(* Logix 5000 project; controller WWTP_SEC_CLX vendor 1 type 14 code 54 rev 17.2; software revision 17.00; part 10 of 13 *)
(* tags used below, declared in another part *)
   Inp_SpeedFdbk : INT;   // Speed Feedbak in Drive Units (typ. 0-32767 = 0 to max freq.)
   Inp_Datalink : INT;   // Auxiliary Signal (datalink) Input in Drive (raw) Units
   Inp_Ready : BOOL;   // 1=Drive is ready to run
   Inp_CommandDir : BOOL;   // 1=Drive is commanded Forward, 0=Drive is commanded Reverse
   Inp_ActualDir : BOOL;   // 1=Drive is running Forward, 0=Drive is running Reverse
   Inp_Accelerating : BOOL;   // 1=Drive is accelerating
   Inp_Decelerating : BOOL;   // 1=Drive is decelerating
   Inp_Alarm : BOOL;   // 1=Drive has an Alarm Condition (see drive display or manual)
   Inp_Faulted : BOOL;   // 1=Drive has Faulted (see drive display or manual)
   Inp_AtSpeed : BOOL;   // 1=Drive is at commanded speed
   Inp_FwdPermOK : BOOL;   // 1=Permissives OK, drive can start Forward
   Inp_FwdNBPermOK : BOOL;   // 1=Non-Bypassable Permissives OK, drive can start Forward
   Inp_RevPermOK : BOOL;   // 1=Permissives OK, drive can start Reverse
   Inp_RevNBPermOK : BOOL;   // 1=Non-Bypassable Permissives OK, motor can start Reverse
   Inp_IntlkOK : BOOL;   // 1=Interlocks OK, drive can start/run
   Inp_NBIntlkOK : BOOL;   // 1=Non-Bypassable Interlocks OK, drive can start/run
   Inp_IOFault : BOOL;   // Input Communication Status 0=OK, 1=fail
   Inp_Sim : BOOL;   // 1=Simulate working drive; 0=Start/Stop/ Monitor actual drive
   Cfg_HasReverse : BOOL;   // 1=Drive can be run reverse, 0=Forward only
   Cfg_HasJog : BOOL;   // 1=Drive Jog Command enabled/visible, 0=Drive Jog Command not allowed
   Cfg_UseRunFdbk : BOOL;   // 1=Drive run feedback should be used for failure checking
   Cfg_HasInpDatalink : BOOL;   // 1=A signal is connected to Inp_Datalink1
   Cfg_HasOutDatalink : BOOL;   // 1=A signal is connected to Out_Datalink1
   Cfg_SetTrack : BOOL;   // 1=PSets track OSets in Oper, OSets track PSets in Prog, 0=no tracking
   Cfg_SetTrackOvrdHand : BOOL;   // 1=Prog/Oper Settings track Override/Hand speed reference
   Cfg_PCmdClear : BOOL;   // 1=Clear Program Commands on receipt 0=Leave Set
   Cfg_SpeedFdbkRawMin : INT;   // Speed Feedback Minimum in Drive (raw) Units (for scaling)
   Cfg_SpeedFdbkRawMax : INT;   // Speed Feedback Maximum in Drive (raw) Units (for scaling)
   Cfg_SpeedFdbkEUMin : REAL;   // Speed Feedback Minimum in Engineering Units (for scaling)
   Cfg_SpeedFdbkEUMax : REAL;   // Speed Feedback Maximum in Engineering Units (for scaling)
   Cfg_InpDatalinkRawMin : INT;   // Input Datalink Minimum in Drive (raw) Units (for scaling)
   Cfg_InpDatalinkRawMax : INT;   // Input Datalink Maximum in Drive (raw) Units (for scaling)
   Cfg_InpDatalinkEUMin : REAL;   // Input Datalink Minimum in Engineering Units (for scaling)
   Cfg_InpDatalinkEUMax : REAL;   // Input Datalink Maximum in Engineering Units (for scaling)
   PSet_SpeedRef : REAL;   // Program Setting of Speed Reference (EU)
   PSet_Owner : DINT;   // Program Owner Request ID (non-zero) or Release (zero)
   OSet_SpeedRef : REAL;   // Operator Setting of Speed Reference (EU)
   PCmd_Start : BOOL;   // Program Command to Start Drive
   PCmd_Stop : BOOL;   // Program Command to Stop Drive
   PCmd_Fwd : BOOL;   // Program Command to set direction to Fowrard
   PCmd_Rev : BOOL;   // Program Command to set direction to Reverse
   PCmd_Acq : BOOL;   // Program Command to Acquire ownership (Oper/OOS to Prog)
   PCmd_Rel : BOOL;   // Program Command to Release ownership (Prog to OOS)
   PCmd_Lock : BOOL;   // Program Command to Lock Mode in Prog
   PCmd_Unlock : BOOL;   // Program Command to Unlock Mode
   PCmd_Reset : BOOL;   // Program Command to Reset drive fault and all Alarms requiring Reset
   PCmd_FailToStartInhibit : BOOL;   // Program Command to Inhibit Fail to Start Alarm
   PCmd_FailToStartUninhibit : BOOL;   // Program Command to Uninhibit Fail to Start Alarm
   PCmd_FailToStopInhibit : BOOL;   // Program Command to Inhibit Fail to Stop Alarm
   PCmd_FailToStopUninhibit : BOOL;   // Program Command to Uninhibit Fail to Stop Alarm
   PCmd_IntlkTripInhibit : BOOL;   // Program Command to Inhibit Interlock Trip Alarm
   PCmd_IntlkTripUninhibit : BOOL;   // Program Command to Uninhibit Interlock Trip Alarm
   PCmd_DriveFaultInhibit : BOOL;   // Program Command to Inhibit Drive Fault Alarm
   PCmd_DriveFaultUninhibit : BOOL;   // Program Command to Uninhibit Drive Fault Alarm
   PCmd_IOFaultInhibit : BOOL;   // Program Command to Inhibit I/O Fault Alarm
   PCmd_IOFaultUninhibit : BOOL;   // Program Command to Uninhibit I/O Fault Alarm
   OCmd_Start : BOOL;   // Operator Command to Start Drive
   OCmd_Stop : BOOL;   // Operator Command to Stop Drive
   OCmd_Jog : BOOL;   // Operator Command to Jog Drive (not cleared by P_VSD!)
   OCmd_Fwd : BOOL;   // Operator Command to set direction to Forward
   OCmd_Rev : BOOL;   // Operator Command to set direction to Reverse
   OCmd_Bypass : BOOL;   // Operator Command to Bypass all Bypassable Interlocks and Permissives
   OCmd_Check : BOOL;   // Operator Command to Check (not bypass) all Interlocks and Permissives
   MCmd_Disable : BOOL;   // Maintenance Command to Disable Drive
   MCmd_Enable : BOOL;   // Maintenance Command to Enable (allow to run) Drive
   OCmd_Reset : BOOL;   // Operator Command to Reset all Alarms requiring Reset
   Val_SpeedRef : REAL;   // Speed Reference (target) to drive
   Val_SpeedFdbk : REAL;   // Speed Feedback (actual) from drive
   Val_InpDatalink : REAL;   // Input Datalink value from drive
   Val_OutDatalink : REAL;   // Output Datalink value to drive
   Val_SpeedFdbkEUMin : REAL;   // Minimum of Speed Feedback = MIN (Cfg_SpeedFdbkEUMin, Cfg_SpeedFdbkEUMax)
   Val_SpeedFdbkEUMax : REAL;   // Maximum of Speed Feedback = MAX (Cfg_SpeedFdbkEUMin, Cfg_SpeedFdbkEUMax)
   Val_Owner : DINT;   // Current Object Owner ID (0=not owned)
   Val_Notify : SINT;   // Current Alarm Level and Acknowledgement (enumeration)
   Sts_Stopped : BOOL;   // 1=Drive requested to stop and is confirmed stopped
   Sts_Starting : BOOL;   // 1=Drive requested to run and awaiting run feedback
   Sts_Running : BOOL;   // 1=Drive requested to run and is confirmed running
   Sts_Stopping : BOOL;   // 1=Drive requested to stop and awaiting stopped feedback
   Sts_Jogging : BOOL;   // 1=Drive requested to Jog
   Sts_CommandDir : BOOL;   // 1=Drive commanded to Forward, 0=Reverse
   Sts_ActualDir : BOOL;   // 1=Drive Actual direction is Forward, 0=Reverse
   Sts_Accel : BOOL;   // 1=Drive is Accelerating
   Sts_Decel : BOOL;   // 1=Drive is Decelerating
   Sts_NotReady : BOOL;   // 1=Drive is Not Ready (cannot be started) Check alarms, stops, faults
   Sts_Alarm : BOOL;   // 1=Drive has an Alarm (see drive display or manual)
   Sts_AtSpeed : BOOL;   // 1=Drive is running at reference speed
   Sts_Available : BOOL;   // 1=Drive available for control by automation (Prog)
   Sts_Bypass : BOOL;   // 1=Bypassable Interlocks and Permissives are Bypassed
   Sts_Disabled : BOOL;   // 1=Drive is Disabled
   Sts_Hand : BOOL;   // 1=Mode is Hand (supersedes Maint, Ovrd, Prog, Oper)
   Sts_Maint : BOOL;   // 1=Mode is Maintenance (supersedes Ovrd, Prog, Oper)
   Sts_Ovrd : BOOL;   // 1=Mode is Override (supersedes Prog, Oper)
   Sts_Prog : BOOL;   // 1=Mode is Program (auto)
   Sts_Oper : BOOL;   // 1=Mode is Operator (manual)
   Sts_FailToStop : BOOL;   // 1=Drive Failed to Stop
   Rdy_Start : BOOL;   // 1=Ready to receive OCmd_Start (enables HMI button)
   Rdy_Stop : BOOL;   // 1=Ready to receive OCmd_Stop (enables HMI button)
   Rdy_Jog : BOOL;   // 1=Ready to receive OCmd_Jog (enables HMI button)
   Rdy_Fwd : BOOL;   // 1=Ready to receive OCmd_Fwd (enabled HMI button)
   Rdy_Rev : BOOL;   // 1=Ready to receive OCmd_Rev (enables HMI button)
   Rdy_Bypass : BOOL;   // 1=Ready to receive OCmd_Bypass (enables HMI button)
   Rdy_Check : BOOL;   // 1=Ready to receive OCmd_Check (enables HMI button)
   Rdy_Disable : BOOL;   // 1=Ready to receive MCmd_Disable (enables HMI button)
   Rdy_Enable : BOOL;   // 1=Ready to receive MCmd_Enable (enables HMI button)
   Rdy_Reset : BOOL;   // 1=Ready to receive OCmd_Reset (enables HMI button)
   Mode : P_Mode;   // Drive Mode Selection
   IOFault : P_Alarm;   // I/O Fault Alarm
   IntlkTrip : P_Alarm;   // Interlock Trip Alarm
   FailToStop : P_Alarm;   // Drive Failed to Stop Alarm
   FailToStart : P_Alarm;   // Drive Failed to Start Alarm
   Wrk_Run : BOOL;   // 1=Drive should be "running", 0=should be "stopped"
   Wrk_AccelT : TIMER;   // Simulation Accel Ramp timer until Running at speed
   Wrk_Fault : BOOL;   // 1=any Fault has been detected
   Wrk_DecelT : TIMER;   // Simulation Decel Ramp time until fully stopped
   Wrk_RunFdbk : BOOL;   // Run Feedback based on mode, simulation, etc. 1=running
   Wrk_Notify : DINT;   // Buffer for building Val_Notify
   Wrk_Bypass : BOOL;   // Internal Bypassable Permissives and Interlocks are Bypassed flag
   Wrk_Disabled : BOOL;   // Internal Drive is Disabled
   DriveFault : P_Alarm;   // Drive Faulted Alarm
   Wrk_SpeedRef : REAL;   // Working copy of Speed Reference (for limiting)
   Wrk_Rev : BOOL;   // Working (internal) Direction 1=Reverse 0=Forward (default)
   Wrk_Jog : BOOL;   // 1=Jog Drive, 0=Drive not jogging
   Wrk_OutDatalink : REAL;   // Selected Output Datalink setting
(* P_VSD, continued *)

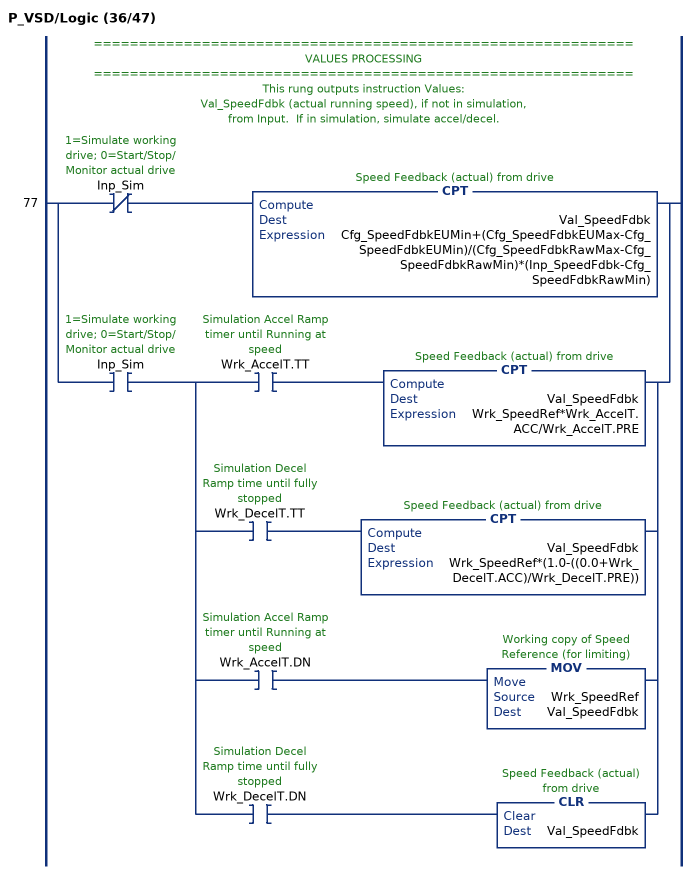
   // ============================================================
   // VALUES PROCESSING
   // ============================================================
   // This rung outputs instruction Values:
   // Val_SpeedFdbk (actual running speed), if not in simulation,
   // from Input.  If in simulation, simulate accel/decel.
   77: [XIO(Inp_Sim) CPT(Val_SpeedFdbk,Cfg_SpeedFdbkEUMin+(Cfg_SpeedFdbkEUMax-Cfg_SpeedFdbkEUMin)/(Cfg_SpeedFdbkRawMax-Cfg_SpeedFdbkRawMin)*(Inp_SpeedFdbk-Cfg_SpeedFdbkRawMin)) ,XIC(Inp_Sim) [XIC(Wrk_AccelT.TT) CPT(Val_SpeedFdbk,Wrk_SpeedRef*Wrk_AccelT.ACC/Wrk_AccelT.PRE) ,XIC(Wrk_DecelT.TT) CPT(Val_SpeedFdbk,Wrk_SpeedRef*(1.0-((0.0+Wrk_DecelT.ACC)/Wrk_DecelT.PRE))) ,XIC(Wrk_AccelT.DN) MOV(Wrk_SpeedRef,Val_SpeedFdbk) ,XIC(Wrk_DecelT.DN) CLR(Val_SpeedFdbk) ] ];
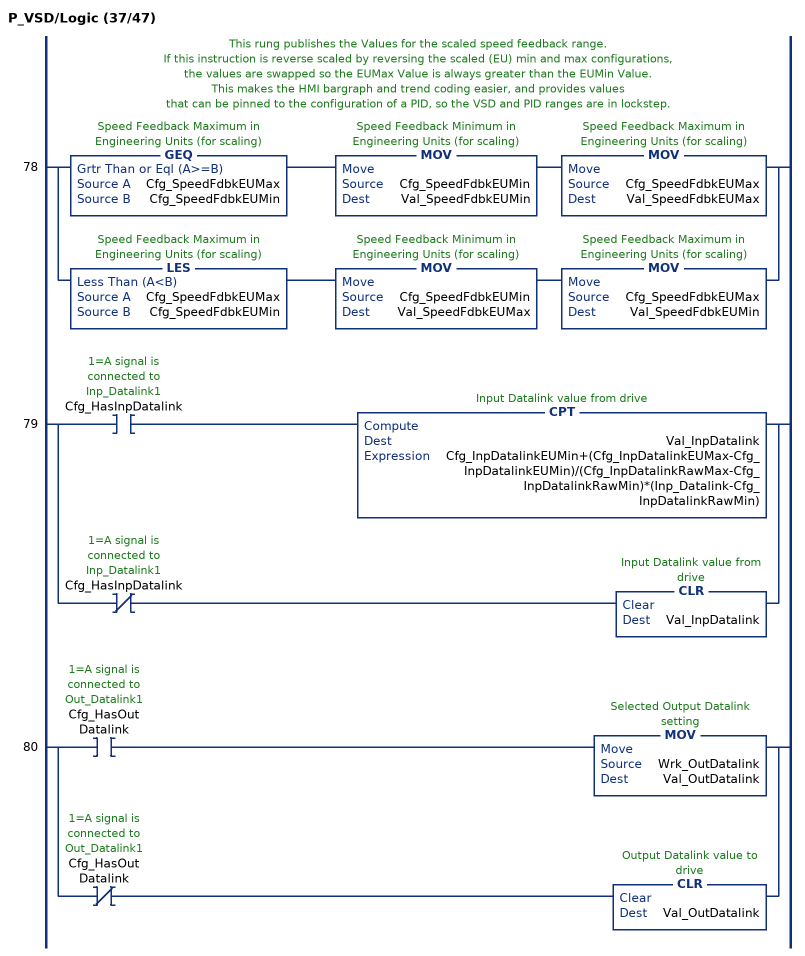
   // This rung publishes the Values for the scaled speed feedback range.
   // If this instruction is reverse scaled by reversing the scaled (EU) min and max configurations,
   // the values are swapped so the EUMax Value is always greater than the EUMin Value.
   // This makes the HMI bargraph and trend coding easier, and provides values
   // that can be pinned to the configuration of a PID, so the VSD and PID ranges are in lockstep.
   78: [GEQ(Cfg_SpeedFdbkEUMax,Cfg_SpeedFdbkEUMin) MOV(Cfg_SpeedFdbkEUMin,Val_SpeedFdbkEUMin) MOV(Cfg_SpeedFdbkEUMax,Val_SpeedFdbkEUMax) ,LES(Cfg_SpeedFdbkEUMax,Cfg_SpeedFdbkEUMin) MOV(Cfg_SpeedFdbkEUMin,Val_SpeedFdbkEUMax) MOV(Cfg_SpeedFdbkEUMax,Val_SpeedFdbkEUMin) ];
   79: [XIC(Cfg_HasInpDatalink) CPT(Val_InpDatalink,Cfg_InpDatalinkEUMin+(Cfg_InpDatalinkEUMax-Cfg_InpDatalinkEUMin)/(Cfg_InpDatalinkRawMax-Cfg_InpDatalinkRawMin)*(Inp_Datalink-Cfg_InpDatalinkRawMin)) ,XIO(Cfg_HasInpDatalink) CLR(Val_InpDatalink) ];
   80: [XIC(Cfg_HasOutDatalink) MOV(Wrk_OutDatalink,Val_OutDatalink) ,XIO(Cfg_HasOutDatalink) CLR(Val_OutDatalink) ];
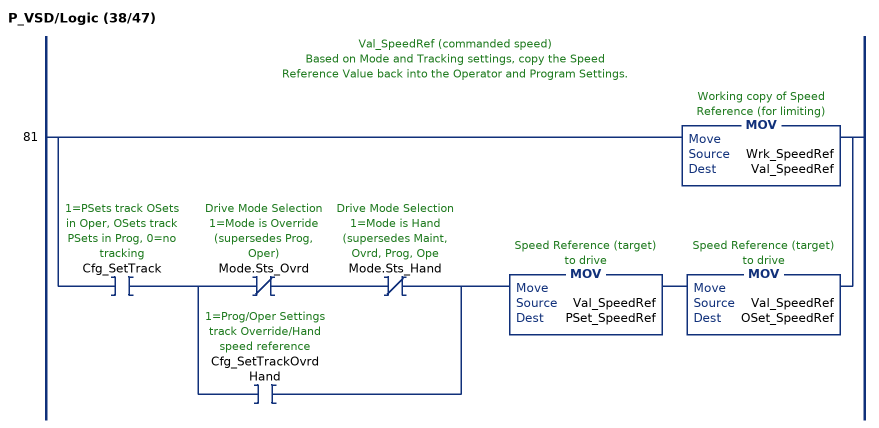
   // Val_SpeedRef (commanded speed)
   // Based on Mode and Tracking settings, copy the Speed
   // Reference Value back into the Operator and Program Settings.
   81: [MOV(Wrk_SpeedRef,Val_SpeedRef) ,XIC(Cfg_SetTrack) [XIO(Mode.Sts_Ovrd) XIO(Mode.Sts_Hand) ,XIC(Cfg_SetTrackOvrdHand) ] MOV(Val_SpeedRef,PSet_SpeedRef) MOV(Val_SpeedRef,OSet_SpeedRef) ];
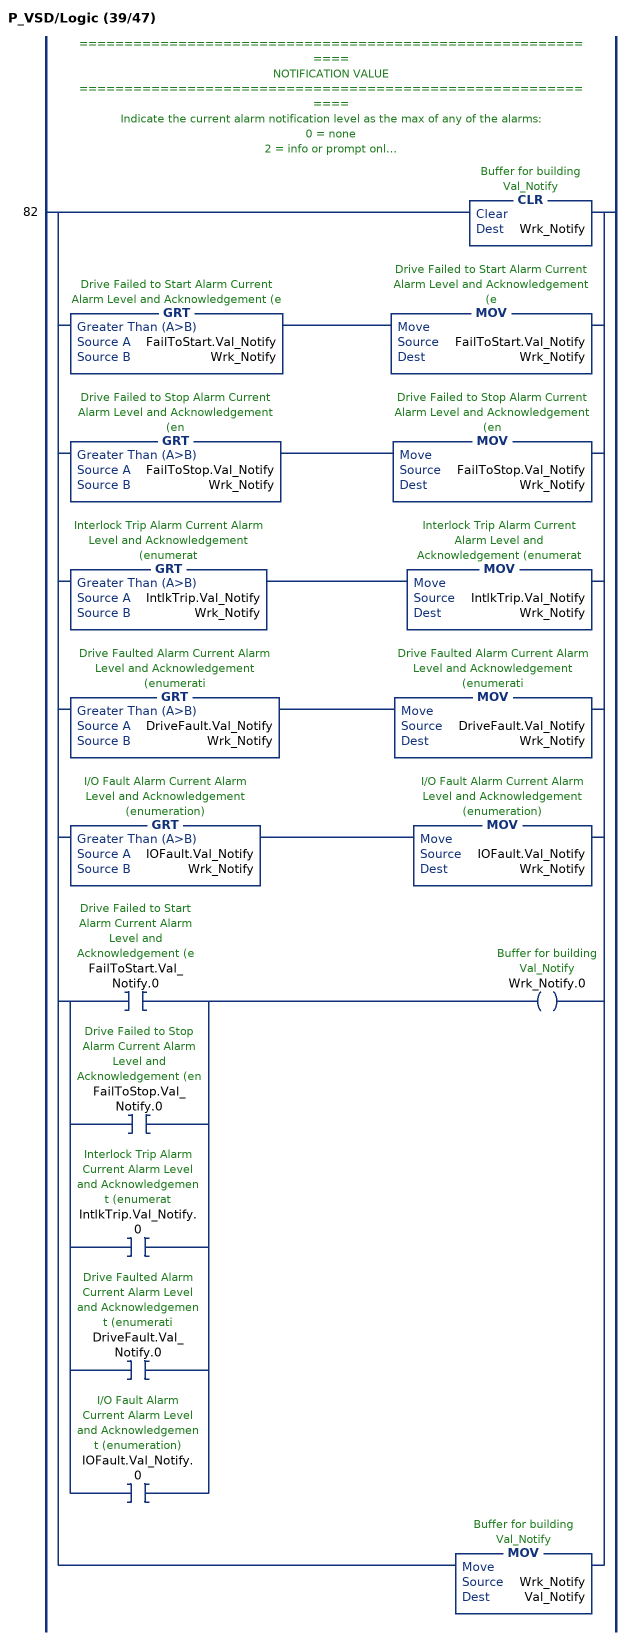
   // ============================================================
   // NOTIFICATION VALUE
   // ============================================================
   // Indicate the current alarm notification level as the max of any of the alarms:
   // 0 = none
   // 2 = info or prompt only
   // 4 = warning
   // 6 = exception (equipment impact)
   // 8 = fault (equipment failure)
   // Add one for any unsuppressed alarm that is not acknowledged (for blink).
   82: [CLR(Wrk_Notify) ,GRT(FailToStart.Val_Notify,Wrk_Notify) MOV(FailToStart.Val_Notify,Wrk_Notify) ,GRT(FailToStop.Val_Notify,Wrk_Notify) MOV(FailToStop.Val_Notify,Wrk_Notify) ,GRT(IntlkTrip.Val_Notify,Wrk_Notify) MOV(IntlkTrip.Val_Notify,Wrk_Notify) ,GRT(DriveFault.Val_Notify,Wrk_Notify) MOV(DriveFault.Val_Notify,Wrk_Notify) ,GRT(IOFault.Val_Notify,Wrk_Notify) MOV(IOFault.Val_Notify,Wrk_Notify) ,[XIC(FailToStart.Val_Notify.0) ,XIC(FailToStop.Val_Notify.0) ,XIC(IntlkTrip.Val_Notify.0) ,XIC(DriveFault.Val_Notify.0) ,XIC(IOFault.Val_Notify.0) ] OTE(Wrk_Notify.0) ,MOV(Wrk_Notify,Val_Notify) ];
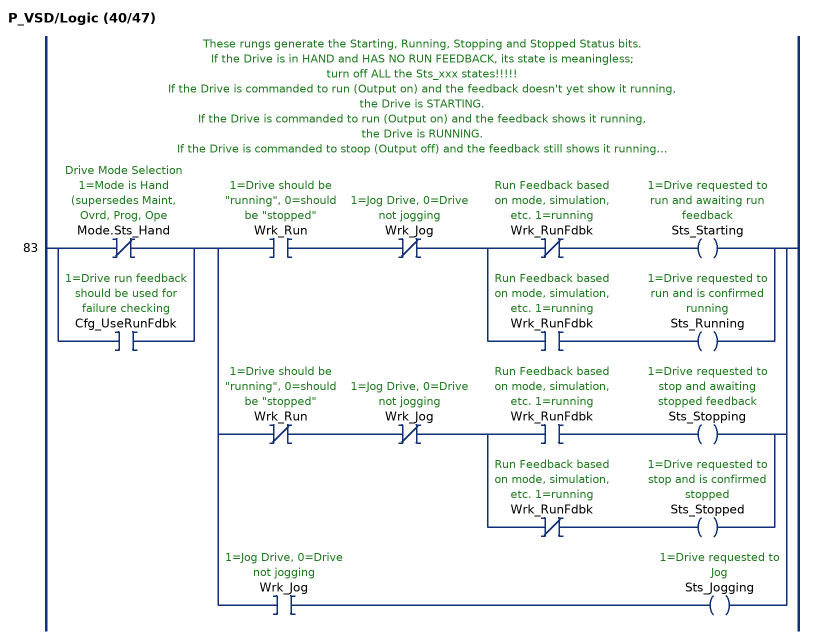
   // These rungs generate the Starting, Running, Stopping and Stopped Status bits.
   // If the Drive is in HAND and HAS NO RUN FEEDBACK, its state is meaningless;
   // turn off ALL the Sts_xxx states!!!!!
   // If the Drive is commanded to run (Output on) and the feedback doesn't yet show it running,
   // the Drive is STARTING.
   // If the Drive is commanded to run (Output on) and the feedback shows it running,
   // the Drive is RUNNING.
   // If the Drive is commanded to stoop (Output off) and the feedback still shows it running,
   // the Drive is STOPPING.
   // If the Drive is commanded to stop (Output off) and the feedback shows it has stopped,
   // the Drive is STOPPED.
   83: [XIO(Mode.Sts_Hand) ,XIC(Cfg_UseRunFdbk) ][XIC(Wrk_Run) XIO(Wrk_Jog) [XIO(Wrk_RunFdbk) OTE(Sts_Starting) ,XIC(Wrk_RunFdbk) OTE(Sts_Running) ] ,XIO(Wrk_Run) XIO(Wrk_Jog) [XIC(Wrk_RunFdbk) OTE(Sts_Stopping) ,XIO(Wrk_RunFdbk) OTE(Sts_Stopped) ] ,XIC(Wrk_Jog) OTE(Sts_Jogging) ];
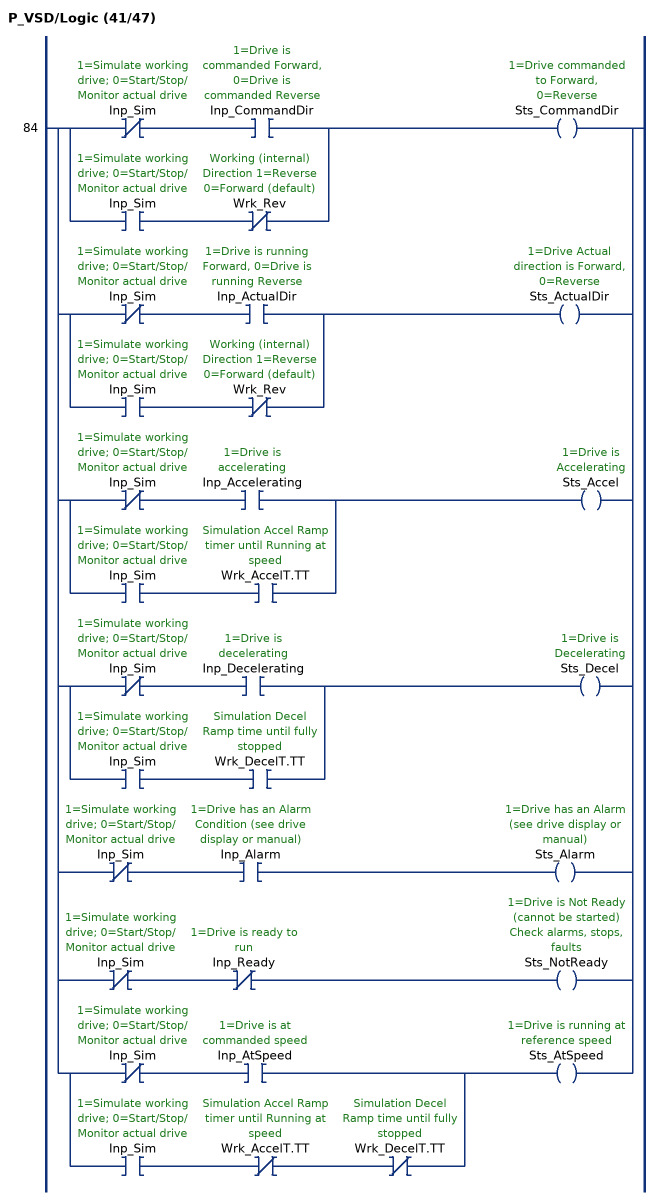
   84: [[XIO(Inp_Sim) XIC(Inp_CommandDir) ,XIC(Inp_Sim) XIO(Wrk_Rev) ] OTE(Sts_CommandDir) ,[XIO(Inp_Sim) XIC(Inp_ActualDir) ,XIC(Inp_Sim) XIO(Wrk_Rev) ] OTE(Sts_ActualDir) ,[XIO(Inp_Sim) XIC(Inp_Accelerating) ,XIC(Inp_Sim) XIC(Wrk_AccelT.TT) ] OTE(Sts_Accel) ,[XIO(Inp_Sim) XIC(Inp_Decelerating) ,XIC(Inp_Sim) XIC(Wrk_DecelT.TT) ] OTE(Sts_Decel) ,XIO(Inp_Sim) XIC(Inp_Alarm) OTE(Sts_Alarm) ,XIO(Inp_Sim) XIO(Inp_Ready) OTE(Sts_NotReady) ,[XIO(Inp_Sim) XIC(Inp_AtSpeed) ,XIC(Inp_Sim) XIO(Wrk_AccelT.TT) XIO(Wrk_DecelT.TT) ] OTE(Sts_AtSpeed) ];
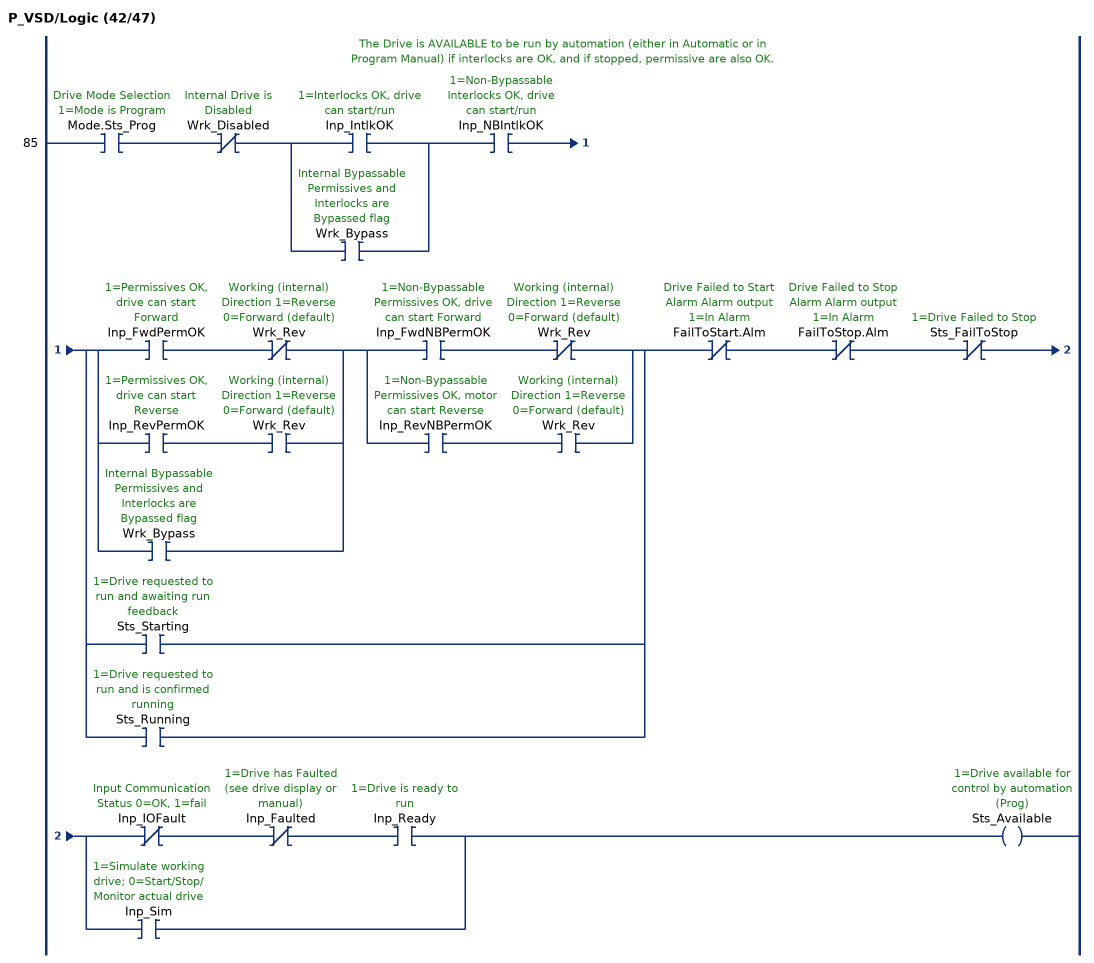
   // The Drive is AVAILABLE to be run by automation (either in Automatic or in
   // Program Manual) if interlocks are OK, and if stopped, permissive are also OK.
   85: XIC(Mode.Sts_Prog)XIO(Wrk_Disabled)[XIC(Inp_IntlkOK) ,XIC(Wrk_Bypass) ]XIC(Inp_NBIntlkOK)[[XIC(Inp_FwdPermOK) XIO(Wrk_Rev) ,XIC(Inp_RevPermOK) XIC(Wrk_Rev) ,XIC(Wrk_Bypass) ] [XIC(Inp_FwdNBPermOK) XIO(Wrk_Rev) ,XIC(Inp_RevNBPermOK) XIC(Wrk_Rev) ] ,XIC(Sts_Starting) ,XIC(Sts_Running) ]XIO(FailToStart.Alm)XIO(FailToStop.Alm)XIO(Sts_FailToStop)[XIO(Inp_IOFault) XIO(Inp_Faulted) XIC(Inp_Ready) ,XIC(Inp_Sim) ]OTE(Sts_Available);
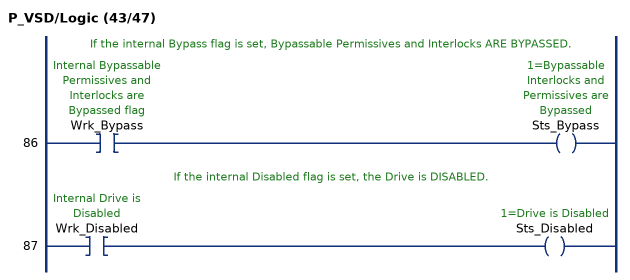
   // If the internal Bypass flag is set, Bypassable Permissives and Interlocks ARE BYPASSED.
   86: XIC(Wrk_Bypass)OTE(Sts_Bypass);
   // If the internal Disabled flag is set, the Drive is DISABLED.
   87: XIC(Wrk_Disabled)OTE(Sts_Disabled);
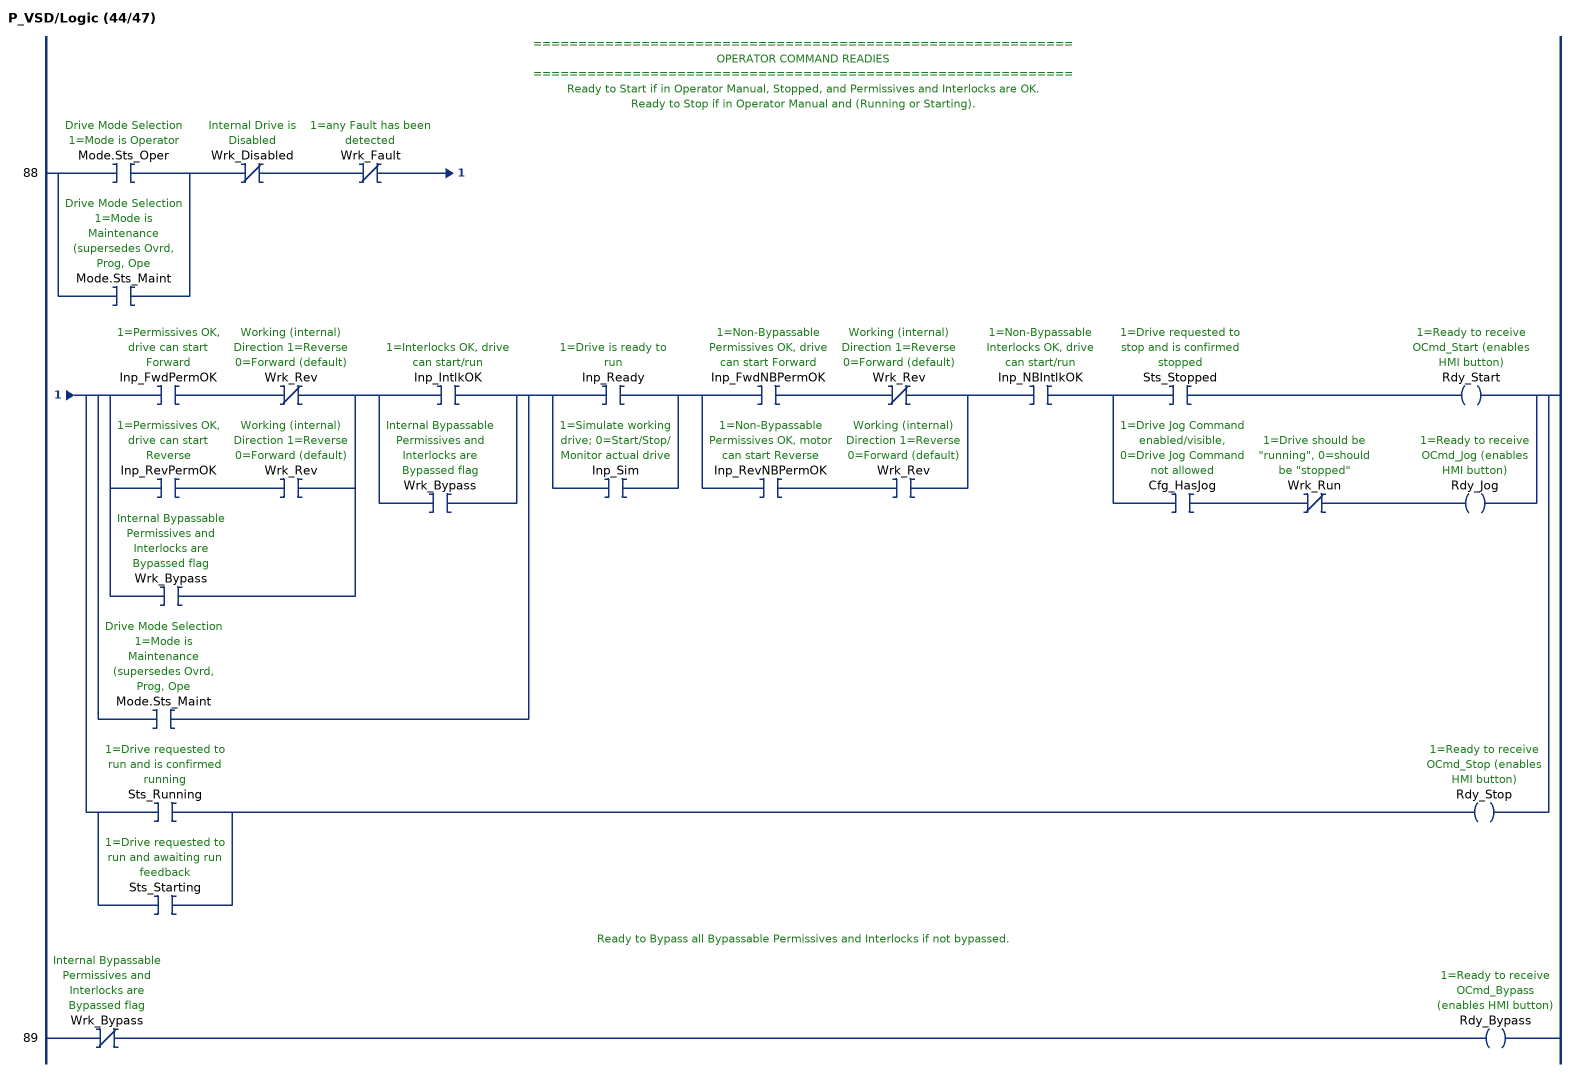
   // ============================================================
   // OPERATOR COMMAND READIES
   // ============================================================
   // Ready to Start if in Operator Manual, Stopped, and Permissives and Interlocks are OK.
   // Ready to Stop if in Operator Manual and (Running or Starting).
   88: [XIC(Mode.Sts_Oper) ,XIC(Mode.Sts_Maint) ]XIO(Wrk_Disabled)XIO(Wrk_Fault)[[[[XIC(Inp_FwdPermOK) XIO(Wrk_Rev) ,XIC(Inp_RevPermOK) XIC(Wrk_Rev) ] ,XIC(Wrk_Bypass) ] [XIC(Inp_IntlkOK) ,XIC(Wrk_Bypass) ] ,XIC(Mode.Sts_Maint) ] [XIC(Inp_Ready) ,XIC(Inp_Sim) ] [XIC(Inp_FwdNBPermOK) XIO(Wrk_Rev) ,XIC(Inp_RevNBPermOK) XIC(Wrk_Rev) ] XIC(Inp_NBIntlkOK) [XIC(Sts_Stopped) OTE(Rdy_Start) ,XIC(Cfg_HasJog) XIO(Wrk_Run) OTE(Rdy_Jog) ] ,[XIC(Sts_Running) ,XIC(Sts_Starting) ] OTE(Rdy_Stop) ];
   // Ready to Bypass all Bypassable Permissives and Interlocks if not bypassed.
   89: XIO(Wrk_Bypass)OTE(Rdy_Bypass);
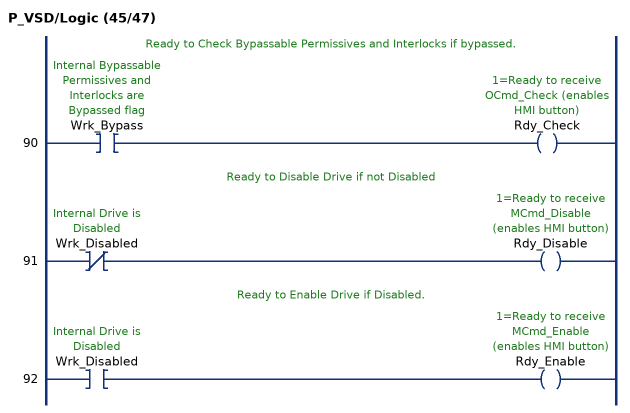
   // Ready to Check Bypassable Permissives and Interlocks if bypassed.
   90: XIC(Wrk_Bypass)OTE(Rdy_Check);
   // Ready to Disable Drive if not Disabled
   91: XIO(Wrk_Disabled)OTE(Rdy_Disable);
   // Ready to Enable Drive if Disabled.
   92: XIC(Wrk_Disabled)OTE(Rdy_Enable);
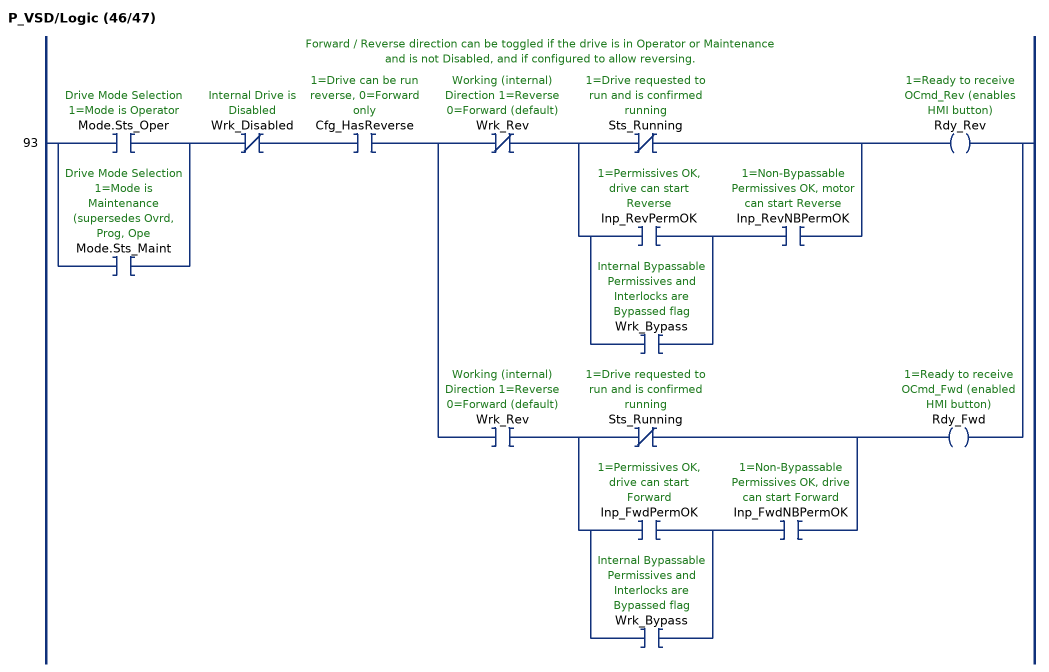
   // Forward / Reverse direction can be toggled if the drive is in Operator or Maintenance
   // and is not Disabled, and if configured to allow reversing.
   93: [XIC(Mode.Sts_Oper) ,XIC(Mode.Sts_Maint) ]XIO(Wrk_Disabled)XIC(Cfg_HasReverse)[XIO(Wrk_Rev) [XIO(Sts_Running) ,[XIC(Inp_RevPermOK) ,XIC(Wrk_Bypass) ] XIC(Inp_RevNBPermOK) ] OTE(Rdy_Rev) ,XIC(Wrk_Rev) [XIO(Sts_Running) ,[XIC(Inp_FwdPermOK) ,XIC(Wrk_Bypass) ] XIC(Inp_FwdNBPermOK) ] OTE(Rdy_Fwd) ];
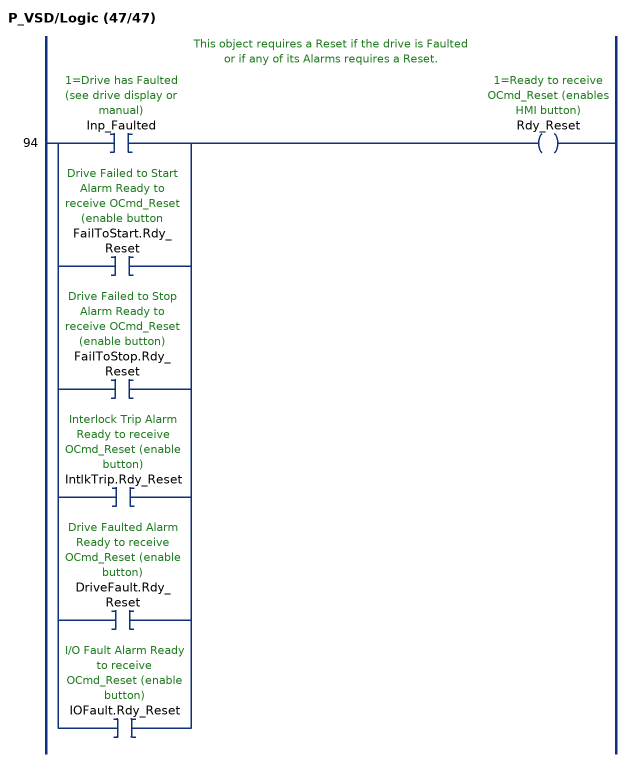
   // This object requires a Reset if the drive is Faulted
   // or if any of its Alarms requires a Reset.
   94: [XIC(Inp_Faulted) ,XIC(FailToStart.Rdy_Reset) ,XIC(FailToStop.Rdy_Reset) ,XIC(IntlkTrip.Rdy_Reset) ,XIC(DriveFault.Rdy_Reset) ,XIC(IOFault.Rdy_Reset) ]OTE(Rdy_Reset);
END_ROUTINE

ROUTINE Prescan   (* ladder *)
// Clear Ownership, set drive to STOP, clear "lurking" Commands
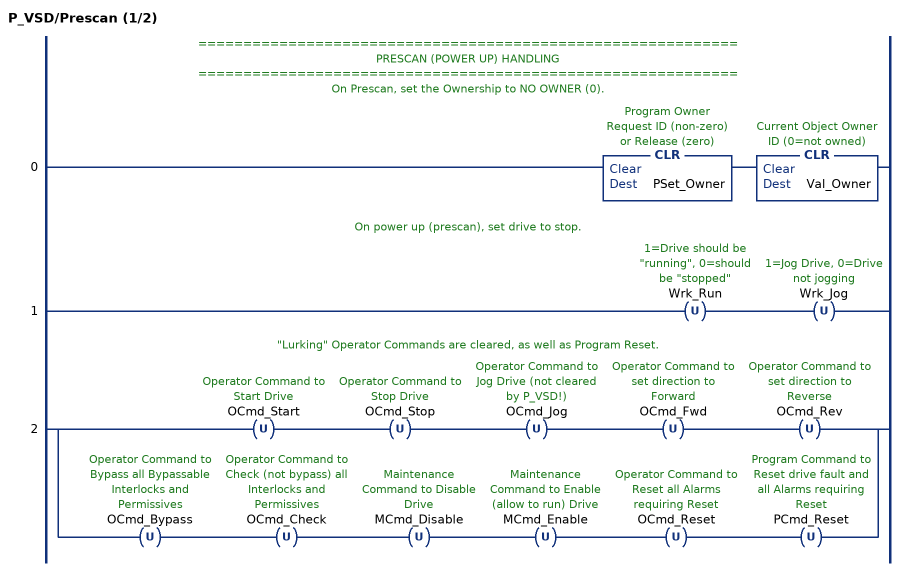
   // ============================================================
   // PRESCAN (POWER UP) HANDLING
   // ============================================================
   // On Prescan, set the Ownership to NO OWNER (0).
   0: CLR(PSet_Owner)CLR(Val_Owner);
   // On power up (prescan), set drive to stop.
   1: OTU(Wrk_Run)OTU(Wrk_Jog);
   // "Lurking" Operator Commands are cleared, as well as Program Reset.
   2: [OTU(OCmd_Start) OTU(OCmd_Stop) OTU(OCmd_Jog) OTU(OCmd_Fwd) OTU(OCmd_Rev) ,OTU(OCmd_Bypass) OTU(OCmd_Check) OTU(MCmd_Disable) OTU(MCmd_Enable) OTU(OCmd_Reset) OTU(PCmd_Reset) ];
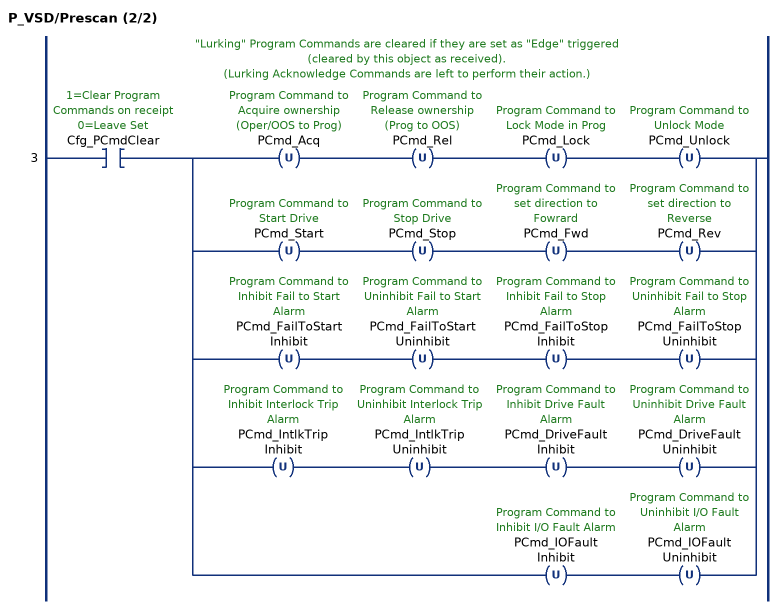
   // "Lurking" Program Commands are cleared if they are set as "Edge" triggered
   // (cleared by this object as received).
   // (Lurking Acknowledge Commands are left to perform their action.)
   3: XIC(Cfg_PCmdClear)[OTU(PCmd_Acq) OTU(PCmd_Rel) OTU(PCmd_Lock) OTU(PCmd_Unlock) ,OTU(PCmd_Start) OTU(PCmd_Stop) OTU(PCmd_Fwd) OTU(PCmd_Rev) ,OTU(PCmd_FailToStartInhibit) OTU(PCmd_FailToStartUninhibit) OTU(PCmd_FailToStopInhibit) OTU(PCmd_FailToStopUninhibit) ,OTU(PCmd_IntlkTripInhibit) OTU(PCmd_IntlkTripUninhibit) OTU(PCmd_DriveFaultInhibit) OTU(PCmd_DriveFaultUninhibit) ,OTU(PCmd_IOFaultInhibit) OTU(PCmd_IOFaultUninhibit) ];
END_ROUTINE
END_ADD_ON_INSTRUCTION

ADD_ON_INSTRUCTION U_CommFail   (* revision 1.0 *)
// Communication Failure Between two PLCs
VAR_INPUT
   Inp_Heartbeat : BOOL; {visible}   // Heartbeat from Remote PLC
   CFG_DelayTimerSec : DINT := 30; {visible}   // Delay Timer in Seconds
END_VAR
VAR_OUTPUT
   Sts_CommFail : BOOL; {visible}   // Communication Failure Alarm
END_VAR
VAR
   HeartBeatDelayTimerOn : TIMER;
   HeartBeatDelayTimerOff : TIMER;
   ConnectionStatusDelayTimer : TIMER;
END_VAR

ROUTINE Logic   (* ladder *)
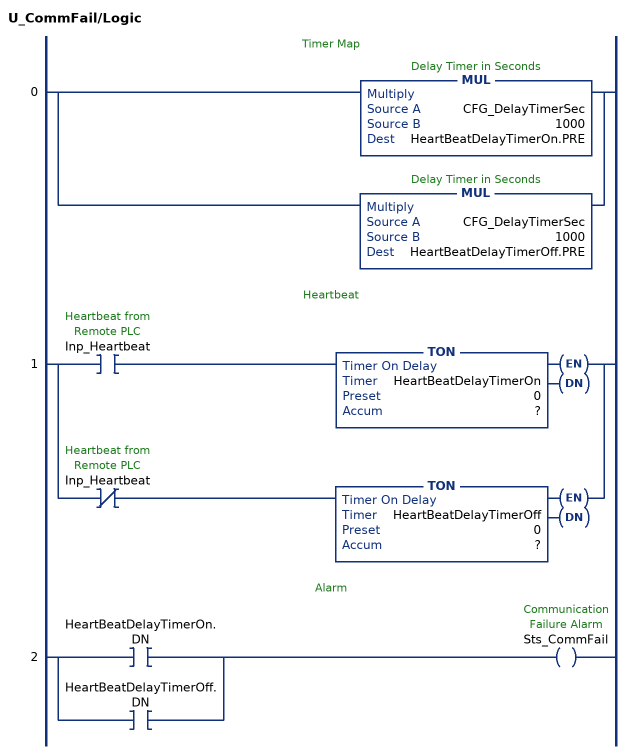
   // Timer Map
   0: [MUL(CFG_DelayTimerSec,1000,HeartBeatDelayTimerOn.PRE) ,MUL(CFG_DelayTimerSec,1000,HeartBeatDelayTimerOff.PRE) ];
   // Heartbeat
   1: [XIC(Inp_Heartbeat) TON(HeartBeatDelayTimerOn,?,?) ,XIO(Inp_Heartbeat) TON(HeartBeatDelayTimerOff,?,?) ];
   // Alarm
   2: [XIC(HeartBeatDelayTimerOn.DN) ,XIC(HeartBeatDelayTimerOff.DN) ]OTE(Sts_CommFail);
END_ROUTINE
END_ADD_ON_INSTRUCTION

ADD_ON_INSTRUCTION U_FlowTot   (* revision 1.0 *)
// Provides Totalization for Daily & Yearly Flow.
VAR_IN_OUT
   Inp_AIn : P_AIn; {required}   // Flow Analog Input AOI
   Inp_WallClock : U_WallClock; {required}   // PLC Wall Clock
END_VAR
VAR_INPUT
   Inp_ProgStartReq : BOOL := 1;   // Prog Start Request. If needed map to turn on totalizer, (ex. pump running) else Defaults to 1 (always start)
END_VAR
VAR_OUTPUT
   Val_FlowRate : REAL; {visible}   // Current Flow Rate
   Val_DailyTot : REAL; {visible}   // Todays Total Flow
   Val_YestTot : REAL; {visible}   // Yesterday Total Flow
   Val_YearlyTot : REAL; {visible}   // This Year Total Flow
   Val_LastYearTot : REAL; {visible}   // Last Year Total Flow
END_VAR
VAR
   YearlyTotalizer : TOTALIZER := (TimeBase := 3, Gain := 1.0, ProgProgReq := 1, ProgStartReq := 1, OperStartReq := 1, RTSTime := 1, ProgOper := 1, RunStop := 1, TargetFlag := 1, TargetDev1Flag := 1, TargetDev2Flag := 1, DeltaT := 0.010000001);
   DailyTotalizer : TOTALIZER := (TimeBase := 3, Gain := 100000.0, ProgStartReq := 1, OperStartReq := 1, RTSTime := 1, ProgOper := 1, RunStop := 1, TargetFlag := 1, TargetDev1Flag := 1, TargetDev2Flag := 1, DeltaT := 0.010000001);
   FlowRateLowLimit_SSUM : SELECTED_SUMMER := (Gain1 := 1.0, Gain2 := 1.0, Gain3 := 1.0, Gain4 := 1.0, Gain5 := 1.0, Gain6 := 1.0, Gain7 := 1.0, Gain8 := 1.0);
   LowCutoff_BNOT : FBD_BOOLEAN_NOT := (In := 1);
   __l00009BB0 : DINT;
   __l00004A73 : REAL;
   __l0000B40A : BOOL;
   __l000041A5 : DINT;
END_VAR

ROUTINE Logic   (* function block diagram *)
   SHEET 1   // Main
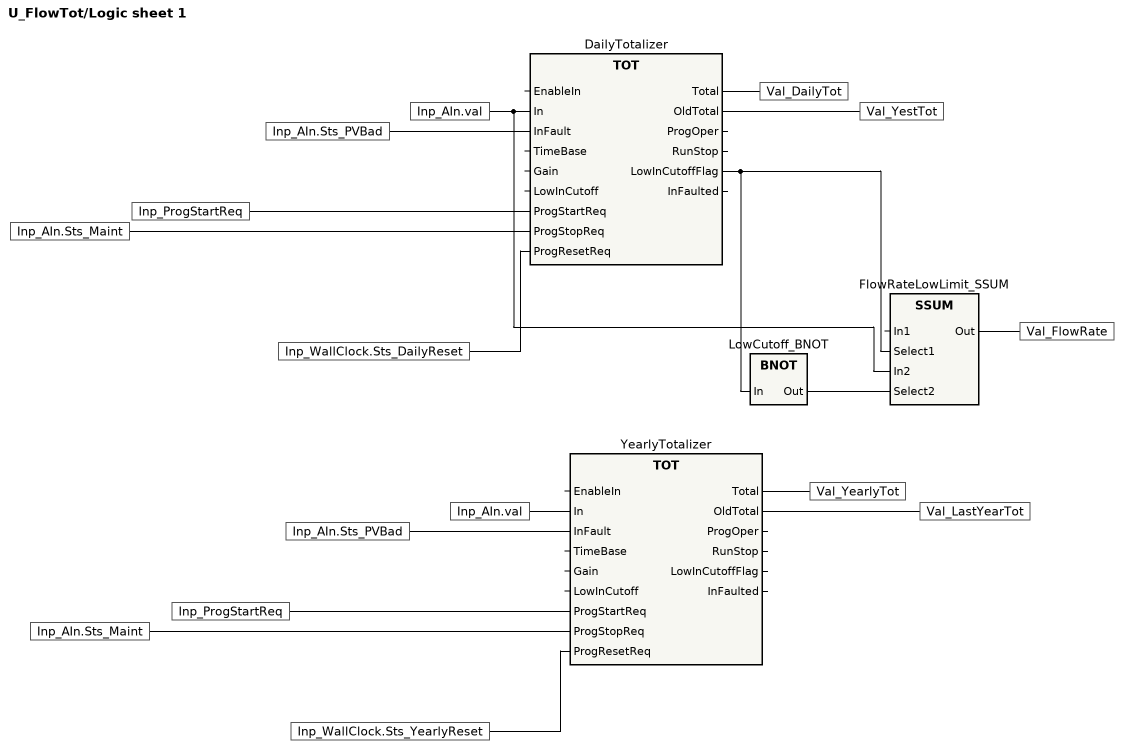
   DailyTotalizer : TOT(In := Inp_AIn.val, InFault := Inp_AIn.Sts_PVBad, ProgStartReq := Inp_ProgStartReq, ProgStopReq := Inp_AIn.Sts_Maint, ProgResetReq := Inp_WallClock.Sts_DailyReset);   // unwired pins: EnableIn TimeBase Gain LowInCutoff ProgOper RunStop InFaulted
   YearlyTotalizer : TOT(In := Inp_AIn.val, InFault := Inp_AIn.Sts_PVBad, ProgStartReq := Inp_ProgStartReq, ProgStopReq := Inp_AIn.Sts_Maint, ProgResetReq := Inp_WallClock.Sts_YearlyReset);   // unwired pins: EnableIn TimeBase Gain LowInCutoff ProgOper RunStop LowInCutoffFlag InFaulted
   LowCutoff_BNOT : BNOT(In := DailyTotalizer.LowInCutoffFlag);
   Val_DailyTot := DailyTotalizer.Total;
   Val_YearlyTot := YearlyTotalizer.Total;
   Val_YestTot := DailyTotalizer.OldTotal;
   FlowRateLowLimit_SSUM : SSUM(Select1 := DailyTotalizer.LowInCutoffFlag, In2 := Inp_AIn.val, Select2 := LowCutoff_BNOT.Out);   // unwired pins: In1
   Val_LastYearTot := YearlyTotalizer.OldTotal;
   Val_FlowRate := FlowRateLowLimit_SSUM.Out;
END_ROUTINE
END_ADD_ON_INSTRUCTION

ADD_ON_INSTRUCTION U_Heartbeat   (* revision 1.0 *)
// Heartbeat Between two PLCs
VAR_INPUT
   CFG_DelayTimerSec : DINT := 30; {visible}   // Delay Timer in Seconds
END_VAR
VAR_OUTPUT
   Heartbeat : BOOL; {visible}   // Heartbeat from Remote PLC
END_VAR
VAR
   DelayTimerOn : TIMER;
   DelayTimerOff : TIMER;
END_VAR

ROUTINE Logic   (* ladder *)
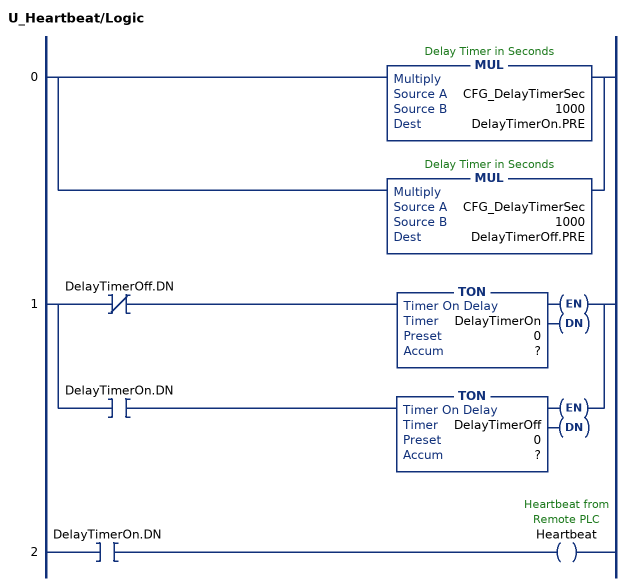
   0: [MUL(CFG_DelayTimerSec,1000,DelayTimerOn.PRE) ,MUL(CFG_DelayTimerSec,1000,DelayTimerOff.PRE) ];
   1: [XIO(DelayTimerOff.DN) TON(DelayTimerOn,?,?) ,XIC(DelayTimerOn.DN) TON(DelayTimerOff,?,?) ];
   2: XIC(DelayTimerOn.DN)OTE(Heartbeat);
END_ROUTINE
END_ADD_ON_INSTRUCTION

ADD_ON_INSTRUCTION U_WallClock   (* revision 1.1 *)
// Wall Clock Set time, Current time and Reset bits.
// Revision note:
// Simplified Day of Week calculation, removed unused tags as a result.
VAR_INPUT
   OCmd_SetTime : BOOL; {visible}   // Set the Date and Time Bit
   OSet_Year : DINT; {visible}   // Year To Set
   OSet_Month : DINT; {visible}   // Month To Set
   OSet_Day : DINT; {visible}   // Day To Set
   OSet_Hour : DINT; {visible}   // Hour To Set
   OSet_Minute : DINT; {visible}   // Minute To Set
   OSet_Second : DINT; {visible}   // Second To Set
END_VAR
VAR_OUTPUT
   Val_CurrentYear : DINT; {visible}   // Current Year
   Val_CurrentMonth : DINT; {visible}   // Current Month
   Val_CurrentDay : DINT; {visible}   // Current Day
   Val_CurrentHour : DINT; {visible}   // Current Hour
   Val_CurrentMinute : DINT; {visible}   // Current Minute
   Val_CurrentSecond : DINT; {visible}   // Current Second
   Val_DayOfWeek : DINT; {visible}   // Day of Week 0 = Sun, 1=Mon, 2=Tues, 3=Wed, 4=Thur, 5=Fri, 6=Sat
   Sts_HourlyReset : BOOL; {visible}   // Hourly Reset
   Sts_DailyReset : BOOL; {visible}   // Daily Reset
   Sts_MonthlyReset : BOOL; {visible}   // Monthly Reset
   Sts_YearlyReset : BOOL; {visible}   // Yearly Reset
END_VAR
VAR
   Wrk_SetDateTime : DINT[7];
   Wrk_GetDateTime : DINT[7];   // Result of GSV to Wallclocktime -- input to Day of Week calculation
        [0]   // Year
        [1]   // Month
        [2]   // Day
        [3]   // Hour
        [4]   // Minute
        [5]   // Second
        [6]   // Microsecond
   Wrk_G : DINT;   // Function of Year and Month, used to calculate Day of Week
   Wrk_F : DINT;   // Function of Month, used to calculate Day of Week
   Wrk_DayONS : BOOL;   // One-Shot for daily pulse output
   Wrk_HourONS : BOOL;   // One-Shot for hourly pulse output
   Wrk_MonthONS : BOOL;   // One-Shot for monthly pulse output
   Wrk_YearONS : BOOL;   // One-Shot for yearly pulse output
END_VAR

ROUTINE Logic   (* ladder *)
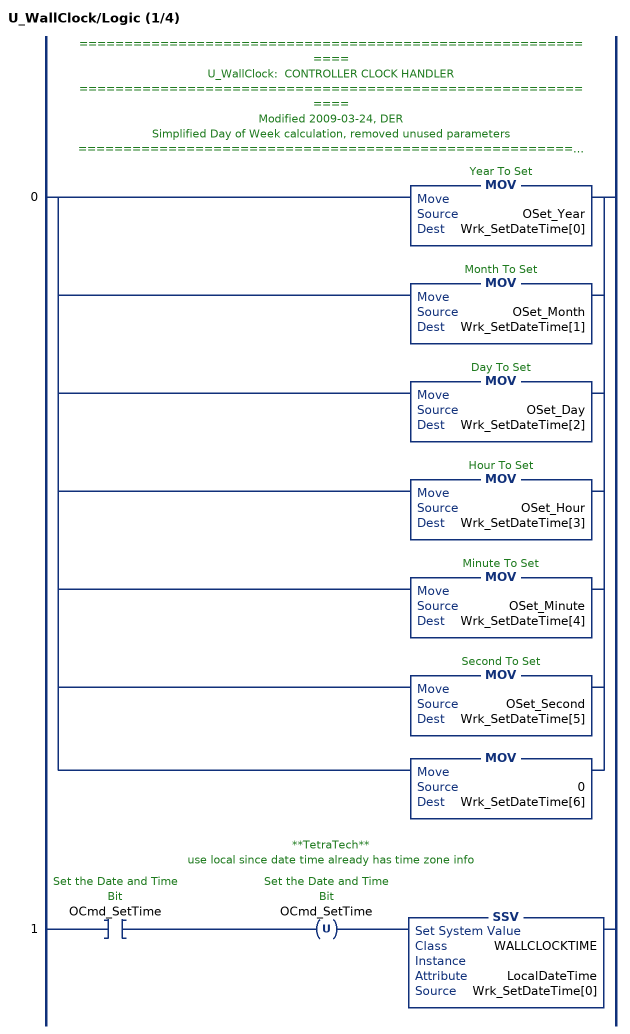
   // ============================================================
   // U_WallClock:  CONTROLLER CLOCK HANDLER
   // ============================================================
   // Modified 2009-03-24, DER
   // Simplified Day of Week calculation, removed unused parameters
   // ============================================================
   // This object manages the controller "Wall Clock", providing date and time services
   // including:
   // * Accepts downloaded date and time and "Set" command from HMI or other sync source and sets the clock
   // * Reads the clock and provides the local date and time to other logic
   // * Calculates and provides the day of the week for the current date
   // * Sets a flag every Hour, Day, Month and Year for resets / data collectors
   // The time is provided as separate Values:
   // Val_CurrentYear : DINT,
   // Val_CurrentMonth : DINT,
   // Val_CurrentDay : DINT,
   // Val_CurrentHour : DINT,
   // Val_CurrentMinute : DINT,
   // Val_CurrentSecond : DINT,
   // Val_DayOfWeek : DINT)
   // ============================================================
   // HANDLE RECEIVED DATE/TIME SYNC, SET CLOCK
   // ============================================================
   // If a date and time have been received with a "Set" command,
   // store the date/time to the controller clock.
   0: [MOV(OSet_Year,Wrk_SetDateTime[0]) ,MOV(OSet_Month,Wrk_SetDateTime[1]) ,MOV(OSet_Day,Wrk_SetDateTime[2]) ,MOV(OSet_Hour,Wrk_SetDateTime[3]) ,MOV(OSet_Minute,Wrk_SetDateTime[4]) ,MOV(OSet_Second,Wrk_SetDateTime[5]) ,MOV(0,Wrk_SetDateTime[6]) ];
   // **TetraTech**
   // use local since date time already has time zone info
   1: XIC(OCmd_SetTime)OTU(OCmd_SetTime)SSV(WALLCLOCKTIME,,LocalDateTime,Wrk_SetDateTime[0]);
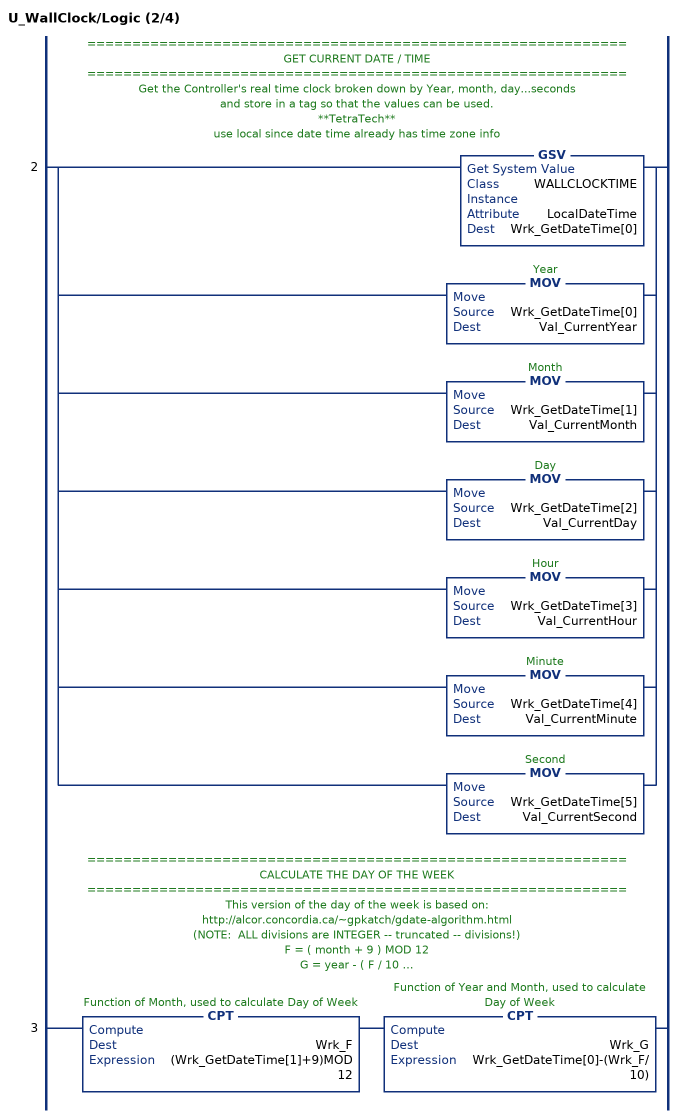
   // ============================================================
   // GET CURRENT DATE / TIME
   // ============================================================
   // Get the Controller's real time clock broken down by Year, month, day...seconds
   // and store in a tag so that the values can be used.
   // **TetraTech**
   // use local since date time already has time zone info
   2: [GSV(WALLCLOCKTIME,,LocalDateTime,Wrk_GetDateTime[0]) ,MOV(Wrk_GetDateTime[0],Val_CurrentYear) ,MOV(Wrk_GetDateTime[1],Val_CurrentMonth) ,MOV(Wrk_GetDateTime[2],Val_CurrentDay) ,MOV(Wrk_GetDateTime[3],Val_CurrentHour) ,MOV(Wrk_GetDateTime[4],Val_CurrentMinute) ,MOV(Wrk_GetDateTime[5],Val_CurrentSecond) ];
   // ============================================================
   // CALCULATE THE DAY OF THE WEEK
   // ============================================================
   // This version of the day of the week is based on:
   // http://alcor.concordia.ca/~gpkatch/gdate-algorithm.html
   // (NOTE:  ALL divisions are INTEGER -- truncated -- divisions!)
   // F = ( month + 9 ) MOD 12
   // G = year - ( F / 10 )
   // Gregorian DayNumber [ D ] = ( 365 * G ) + ( G / 4 ) - ( G / 100 ) + ( G / 400 ) + ( ( ( F * 306 ) + 5 ) / 10 ) + day - 1
   // DayOfWeek = ( DayNumber + 3 ) MOD 7
   // ~~~~~~~~~~~~~~~~~~~~~~~~~~~~~~~~~~~~~~~~~~~~~~~~~~~~~~~~~~~~
   // This rung calculates the "G" and "F" functions shown in the algorithm above.
   // ~~~~~~~~~~~~~~~~~~~~~~~~~~~~~~~~~~~~~~~~~~~~~~~~~~~~~~~~~~~~
   3: CPT(Wrk_F,(Wrk_GetDateTime[1]+9)MOD 12)CPT(Wrk_G,Wrk_GetDateTime[0]-(Wrk_F/10));
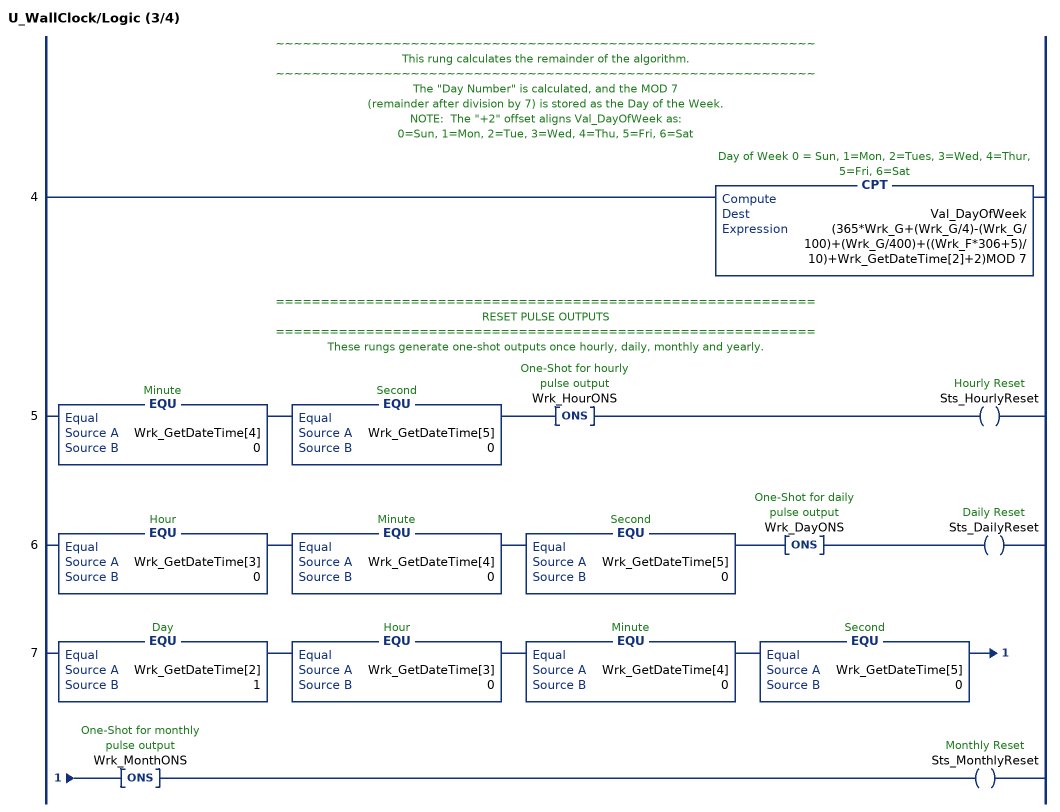
   // ~~~~~~~~~~~~~~~~~~~~~~~~~~~~~~~~~~~~~~~~~~~~~~~~~~~~~~~~~~~~
   // This rung calculates the remainder of the algorithm.
   // ~~~~~~~~~~~~~~~~~~~~~~~~~~~~~~~~~~~~~~~~~~~~~~~~~~~~~~~~~~~~
   // The "Day Number" is calculated, and the MOD 7
   // (remainder after division by 7) is stored as the Day of the Week.
   // NOTE:  The "+2" offset aligns Val_DayOfWeek as:
   // 0=Sun, 1=Mon, 2=Tue, 3=Wed, 4=Thu, 5=Fri, 6=Sat
   4: CPT(Val_DayOfWeek,(365*Wrk_G+(Wrk_G/4)-(Wrk_G/100)+(Wrk_G/400)+((Wrk_F*306+5)/10)+Wrk_GetDateTime[2]+2)MOD 7);
   // ============================================================
   // RESET PULSE OUTPUTS
   // ============================================================
   // These rungs generate one-shot outputs once hourly, daily, monthly and yearly.
   5: EQU(Wrk_GetDateTime[4],0)EQU(Wrk_GetDateTime[5],0)ONS(Wrk_HourONS)OTE(Sts_HourlyReset);
   6: EQU(Wrk_GetDateTime[3],0)EQU(Wrk_GetDateTime[4],0)EQU(Wrk_GetDateTime[5],0)ONS(Wrk_DayONS)OTE(Sts_DailyReset);
   7: EQU(Wrk_GetDateTime[2],1)EQU(Wrk_GetDateTime[3],0)EQU(Wrk_GetDateTime[4],0)EQU(Wrk_GetDateTime[5],0)ONS(Wrk_MonthONS)OTE(Sts_MonthlyReset);
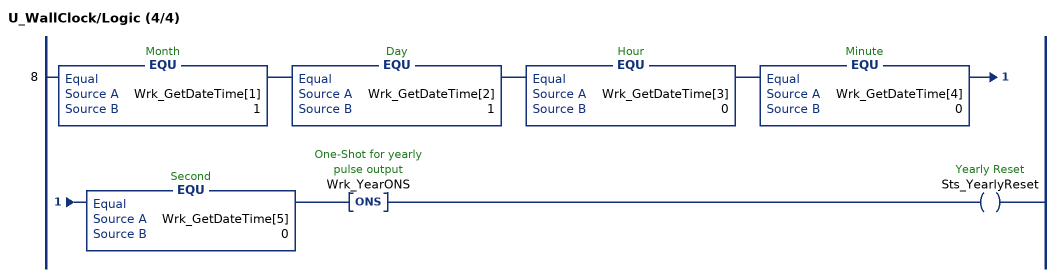
   8: EQU(Wrk_GetDateTime[1],1)EQU(Wrk_GetDateTime[2],1)EQU(Wrk_GetDateTime[3],0)EQU(Wrk_GetDateTime[4],0)EQU(Wrk_GetDateTime[5],0)ONS(Wrk_YearONS)OTE(Sts_YearlyReset);
END_ROUTINE
END_ADD_ON_INSTRUCTION
